INTERFACE I_Process_LinkedList

METHOD AddHeadValue : ST_PROCESS_LIST_RESULT
VAR_INPUT
  stData        : ST_PROCESS_DATA;
END_VAR
END_METHOD

METHOD AddTailValue : ST_PROCESS_LIST_RESULT
VAR_INPUT
  stData        : ST_PROCESS_DATA;
END_VAR
END_METHOD

PROPERTY Count : UDINT
GET
END_GET
END_PROPERTY

PROPERTY Data : ARRAY[1..MAX_LIST_NODES] OF ST_PROCESS_DATA
GET
END_GET
END_PROPERTY

PROPERTY Free : UDINT
GET
END_GET
END_PROPERTY

METHOD GetHead : ST_PROCESS_LIST_RESULT
VAR_INPUT
END_VAR
END_METHOD

METHOD InitList : BOOL
END_METHOD

PROPERTY Nodes : ARRAY[0..MAX_LIST_NODES] OF T_LinkedListEntry
GET
END_GET
END_PROPERTY

METHOD RemoveHeadValue : ST_PROCESS_LIST_RESULT
VAR_INPUT
END_VAR
END_METHOD

END_INTERFACE

(* stored: Version 1.1.0.1
   Itf I_Process_LinkedList: Id {829273fc-f0e4-421e-8e8f-b1ed075e6f00}
   Method AddHeadValue: Id {555d3811-677b-41c6-ae5c-3e3de83d404d}
   Method AddTailValue: Id {45c5b212-8621-4c6e-9784-533e2c004c61}
   Property Count: Id {7f89da67-9649-4854-82b0-55285bbdf36e}
   Get Get: Id {626d5db2-1b35-4988-886f-eb5573e72a13}
   Property Data: Id {b0c21623-a37c-4901-8687-96b7a2f9a9e7}
   Get Get: Id {bd059851-6a09-4f75-aeaf-fd3416fb6557}
   Property Free: Id {68bbda69-0988-4457-b19e-42457a6014e8}
   Get Get: Id {c2bde1fa-a2d9-4af2-a223-e3f33240b24d}
   Method GetHead: Id {dc06304c-71c8-4f34-b570-6515eefadc77}
   Method InitList: Id {567ec93b-00c8-47b4-92f7-fe5fccee77f8}
   Property Nodes: Id {bdee395e-92ed-487b-99c3-9b921440af8b}
   Get Get: Id {226cce63-7092-4773-af55-2cdb2da2692d}
   Method RemoveHeadValue: Id {cdc6830c-ead2-4ea2-b1b0-4d1382816aae} *)
